FUNCTION_BLOCK State_Mockup EXTENDS State
VAR
	_IsExecuting : BOOL;
END_VAR

METHOD Executing : BOOL
_IsExecuting := TRUE;
END_METHOD

PROPERTY IsExecuting : BOOL
GET
IsExecuting := _IsExecuting;
END_GET
END_PROPERTY

END_FUNCTION_BLOCK

(* stored: Version 1.1.0.1, ProductVersion 3.1.4026.18
   POU State_Mockup: Id {40f03ece-c10d-4dae-a4a6-33689633f203}, SpecialFunc None
   Method Executing: Id {d6c45f4c-4622-43f9-894c-25a4eb7ffec9}
   Property IsExecuting: Id {58e32660-0e87-469a-9b53-a3f745ad9b8e}
   Get Get: Id {1cc2c7e6-f010-4e9e-ad36-5e1eee546f33} *)
